DATA_BLOCK "DT-Chars_DB"
{ S7_Optimized_Access := 'FALSE' }
VERSION : 0.1
NON_RETAIN
"DT-Chars"

BEGIN

END_DATA_BLOCK

